// TwinCAT 3 PLC project FirstPLC
// ProgramVersion: 3.1.4024.0
// libraries:
//   Tc2_Standard, * (Beckhoff Automation GmbH)
//   Tc2_System, * (Beckhoff Automation GmbH)
//   Tc3_Module, * (Beckhoff Automation GmbH)
//   TcUnit, * (www.tcunit.org)
// project tree:
//   / PlcTask.TcTTO (not stored), PlcTask2.TcTTO
//   POUs/ FB_TestSuite1.TcPOU (not stored), FB_TestSuite2.TcPOU, FB_TestSuite3.TcPOU, FB_TestSuiteGroup.TcPOU, FB_TestSuite_CFC.TcPOU, MAIN.TcPOU, PRG_TESTS.TcPOU
// real-time tasks:
//   TASK PlcTask: cycle T#10ms, priority 20, ADS port 350
//   TASK PlcTask2: cycle T#10ms, priority 1, ADS port 351

CONFIGURATION FirstPLC
    RESOURCE PLC ON TwinCAT3
        TASK PlcTask2(INTERVAL := T#10ms, PRIORITY := 1);
        PROGRAM PRG_TESTS WITH PlcTask2 : PRG_TESTS;
    END_RESOURCE
END_CONFIGURATION

// ---- POUs/PRG_TESTS.TcPOU
PROGRAM PRG_TESTS
VAR
    fbTestSuite1Instance1 : FB_TestSuite1;
    fbTestSuite2Instance1 : FB_TestSuite2;
    fbTestSuite2Instance2 : FB_TestSuite2;
    fbTestSuiteGroup : FB_TestSuiteGroup;
	fbTestSuiteInstance3_CFC : FB_TestSuite_CFC;
END_VAR

TcUnit.RUN();

END_PROGRAM

// ---- POUs/FB_TestSuite2.TcPOU
FUNCTION_BLOCK FB_TestSuite2 EXTENDS FB_TestSuite
VAR_INPUT
END_VAR
VAR_OUTPUT
END_VAR
VAR
END_VAR

TestCase2A();
TestCase2B();

TEST('TestCase2C');

AssertTrue(TRUE, 'Condition is not true');
AssertTrue(FALSE, 'Condition is not true');

TEST_FINISHED();

METHOD PUBLIC Method_CFC : BOOL
VAR_INPUT
END_VAR
END_METHOD

METHOD PUBLIC Method_FBD : BOOL
VAR_INPUT
END_VAR
// NETWORK 1
END_METHOD

METHOD PUBLIC Method_LD : BOOL
VAR_INPUT
END_VAR
// NETWORK 1
END_METHOD

METHOD TestCase2A
VAR_INPUT
END_VAR
TEST('TestCase2A');

AssertTrue(TRUE, 'Condition is not true');

TEST_FINISHED();
END_METHOD

METHOD TestCase2B
VAR_INPUT
END_VAR
TEST('TestCase2B');

AssertTrue(TRUE, 'Condition is not true');
AssertTrue(TRUE, 'Condition is not true');

TEST_FINISHED();
END_METHOD

END_FUNCTION_BLOCK

// ---- POUs/FB_TestSuiteGroup.TcPOU
FUNCTION_BLOCK FB_TestSuiteGroup
VAR
    fbTestSuite3Instance1 : FB_TestSuite3;
    fbTestSuite3Instance2 : FB_TestSuite3;
END_VAR

END_FUNCTION_BLOCK

// ---- POUs/FB_TestSuite3.TcPOU
FUNCTION_BLOCK FB_TestSuite3 EXTENDS FB_TestSuite
VAR_INPUT
END_VAR
VAR_OUTPUT
END_VAR
VAR
END_VAR

TestCase3A();
TestCase3B();

METHOD TestCase3B
VAR_INPUT
END_VAR
TEST('TestCase3B');

AssertTrue(TRUE, 'Condition is not true');
AssertTrue(TRUE, 'Condition is not true');

TEST_FINISHED();
END_METHOD

METHOD TestCase3A
VAR_INPUT
END_VAR
TEST('TestCase3A');

AssertTrue(TRUE, 'Condition is not true');
AssertTrue(TRUE, 'Condition is not true');

TEST_FINISHED();
END_METHOD

END_FUNCTION_BLOCK

// ---- POUs/FB_TestSuite_CFC.TcPOU
FUNCTION_BLOCK FB_TestSuite_CFC EXTENDS TcUnit.FB_TestSuite
VAR_INPUT
END_VAR
VAR_OUTPUT
END_VAR
VAR
END_VAR

END_FUNCTION_BLOCK

// ---- POUs/MAIN.TcPOU
PROGRAM MAIN
VAR
    bTest : BOOL;
END_VAR

END_PROGRAM
